// TIA Portal V17 export
// export: Created 2025-03-07T09:17:01.5177365Z, ExportSetting WithDefaults, DisplayName Totally Integrated Automation Portal, DisplayVersion V17 Update 8, DisplayName TIA Portal Openness, DisplayVersion V17 Update 8, DisplayName TIA Portal Version Control Interface, DisplayVersion V17, DisplayName SINAMICS Startdrive Advanced, DisplayVersion V17 SP2, DisplayName SINAMICS Startdrive G110M, G120, G120C, G120D, G120P, G115D, DisplayVersion V17 SP2, DisplayName SINAMICS Startdrive G130, G150, S120, S150, SINAMICS MV, S210, DisplayVersion V17 SP2, DisplayName STEP 7 Professional, DisplayVersion V17 Update 8, DisplayName SINUMERIK ONE STEP 7 Toolbox, DisplayVersion V17 Update 12, DisplayName SINUMERIK 840D sl STEP 7 Toolbox, DisplayVersion V17 Update 12, DisplayName STEP 7 Safety, DisplayVersion V17 Update 6, DisplayName WinCC Advanced, DisplayVersion V17 Update 8
FUNCTION "FC7340_POWDER_PLC_INTERLOCK" : Void   // FC7340, LAD
{ S7_Optimized_Access := 'TRUE' }
VERSION : 0.1
// stored: AutoNumber false, IsIECCheckEnabled false, SetENOAutomatically false, UDAEnableTagReadback false
   VAR_TEMP
      INPUTS : HW_IO;
      OUTPUTS : HW_IO;
      RETVAL_FILL : Int;
   END_VAR
BEGIN

REGION Network 1: INPUTS
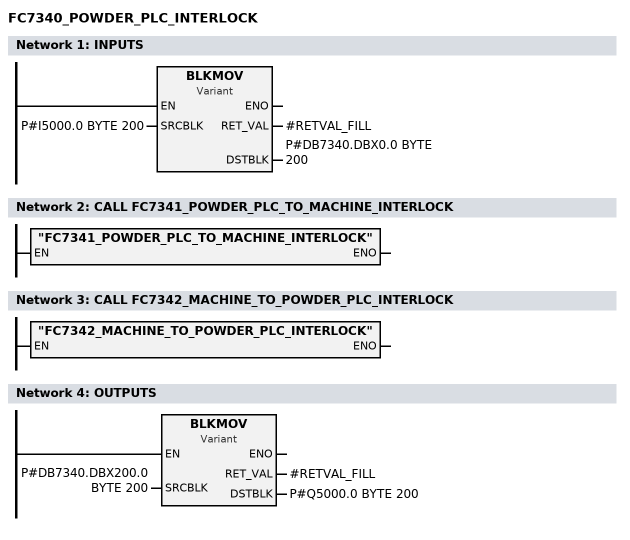
   RUNG wire#powerrail
      { S7_Templates := "blk_type := Variant" } BLKMOV(SRCBLK := P#I5000.0 BYTE 200, RET_VAL => #RETVAL_FILL, DSTBLK => P#DB7340.DBX0.0 BYTE 200)
   END_RUNG
   // the same network as SCL:
   #RETVAL_FILL := BLKMOV(SRCBLK := P#I5000.0 BYTE 200, DSTBLK => P#DB7340.DBX0.0 BYTE 200);
END_REGION

REGION Network 2: CALL FC7341_POWDER_PLC_TO_MACHINE_INTERLOCK
   RUNG wire#powerrail
      "FC7341_POWDER_PLC_TO_MACHINE_INTERLOCK"()
   END_RUNG
   // the same network as SCL:
   "FC7341_POWDER_PLC_TO_MACHINE_INTERLOCK"();
END_REGION

REGION Network 3: CALL FC7342_MACHINE_TO_POWDER_PLC_INTERLOCK
   RUNG wire#powerrail
      "FC7342_MACHINE_TO_POWDER_PLC_INTERLOCK"()
   END_RUNG
   // the same network as SCL:
   "FC7342_MACHINE_TO_POWDER_PLC_INTERLOCK"();
END_REGION

REGION Network 4: OUTPUTS
   RUNG wire#powerrail
      { S7_Templates := "blk_type := Variant" } BLKMOV(SRCBLK := P#DB7340.DBX200.0 BYTE 200, RET_VAL => #RETVAL_FILL, DSTBLK => P#Q5000.0 BYTE 200)
   END_RUNG
   // the same network as SCL:
   #RETVAL_FILL := BLKMOV(SRCBLK := P#DB7340.DBX200.0 BYTE 200, DSTBLK => P#Q5000.0 BYTE 200);
END_REGION
END_FUNCTION
